(*

.. <legal notes>

legal notes
=================
| SPDX-FileCopyrightText: © 2025 Oleksandr Tiutyk <trofimich@gmail.com>
| SPDX-License-Identifier: LGPL-3.0-only
| For details check: LGPL-3.0-only_

.. _LGPL-3.0-only: https://www.gnu.org/licenses/lgpl-3.0.en.html

.. </legal notes>

*)

{attribute 'no_explicit_call' := 'do not call this function block directly'} 
{attribute 'enable_dynamic_creation'}
FUNCTION_BLOCK WhileActivity EXTENDS SequenceActivity IMPLEMENTS IWhileActivity
VAR
	{attribute 'OPC.UA.DA' := '0'}
	_Condition : ICondition;	
END_VAR

{attribute 'monitoring' := 'call'}
PROPERTY ClassName : STRING
GET
ClassName := _ClassName;
END_GET
END_PROPERTY

{attribute 'monitoring' := 'call'}
PROPERTY FINAL Condition : ICondition
GET
Condition := _Condition;
END_GET
SET
_Condition := Condition;
END_SET
END_PROPERTY

METHOD Configure
VAR_INPUT
	condition : ICondition; 
END_VAR
VAR
	argumentNullException : Core.ArgumentNullException;
END_VAR
IF condition = 0 THEN
	argumentNullException.Throw(NamespaceName, ClassName, __POUNAME(), __POSITION(), 'condition');
END_IF

_Condition := condition;
END_METHOD

METHOD FB_init : BOOL
VAR_INPUT
	(* if TRUE, the retain variables are initialized (warm start / cold start)*)
	bInitRetains	: BOOL;
	(* if TRUE, the instance afterwards gets moved into the copy code (online change)*)
	bInCopyCode	: BOOL;
	workflow : IWorkflow;
END_VAR
_ClassName := 'WhileActivity';
END_METHOD

{attribute 'monitoring' := 'call'}
PROPERTY NamespaceName : STRING
GET
NamespaceName := CurrentNamespace.Name;
END_GET
END_PROPERTY

METHOD PROTECTED OnRunning 
VAR_INPUT
	isStart : BOOL;
END_VAR
VAR_OUTPUT
	done : BOOL;
END_VAR
VAR
	workflowVariable : Core.GENERIC_VALUE;
	
	argumentNullException : Core.NullReferenceException;
END_VAR
IF _Condition = 0 THEN
	argumentNullException.Throw(NamespaceName, ClassName, __POUNAME(), __POSITION(), 'Condition');
END_IF

IF isStart THEN
	IF NOT _Condition.Evaluate(THIS^) THEN
		done := TRUE;
		RETURN;
	END_IF
END_IF

SUPER^.OnRunning(isStart, done => done);

IF done THEN
	IF _Condition.Evaluate(THIS^) THEN
		SUPER^.OnRunning(TRUE, done => done);
	ELSE
		done := TRUE;
	END_IF
END_IF
END_METHOD

{attribute 'monitoring' := 'call'}
PROPERTY Size : ULINT
GET
Size := XSIZEOF(THIS^);
END_GET
END_PROPERTY

END_FUNCTION_BLOCK

(* stored: Version 1.1.0.1
   POU WhileActivity: Id {12c9e06e-5895-45ce-9974-6263c896f40b}, SpecialFunc None
   Folder Overriden: Id {8c1d4263-b645-4c82-9dcb-55337470aad6}
   Property ClassName: Id {945e9c30-b95b-43ef-9233-6a843f2d82bf}
   Get Get: Id {3597e220-3046-4e42-8ec4-3ada54f3efb7}
   Property Condition: Id {9ffd553d-7db0-4b59-8a79-f5a38ea8bdc4}
   Get Get: Id {22d12ecc-b75f-4acd-863e-d1c14b62fdde}
   Set Set: Id {43185451-72c8-4e95-941a-bebcb25c083f}
   Method Configure: Id {d5142548-dc1c-407c-a71e-5333193ceff2}
   Method FB_init: Id {6a543e26-62cd-441c-81f4-01e022c2491c}
   Property NamespaceName: Id {abbe54cc-0f22-4490-b6ad-3ab1233e3c46}
   Get Get: Id {b9366bd0-05b4-40cb-8b69-19098e53d90b}
   Method OnRunning: Id {346689b4-fcd7-4614-871f-ef4906187553}
   Property Size: Id {ef186776-ee7b-48a8-9b46-2633dc3274c4}
   Get Get: Id {cfd06962-6fec-4072-a8bc-e00513767b8d} *)
